FUNCTION_BLOCK LogSchedule (* Basic Function Block Type *)
  (* Standard: 61499-2 *)
  (* Version 0.0, 11/2/2016, chivdan, nxtControl GmbH, Template *)
  PACKAGE Main;
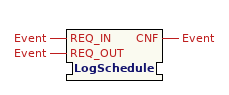
  EVENT_INPUT
    REQ_IN; (* Normal Execution Request *)
    REQ_OUT;
  END_EVENT
  EVENT_OUTPUT
    CNF;
  END_EVENT
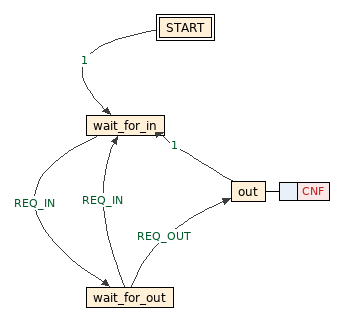
  EC_STATES
    START; (* Initial State *)
    wait_for_in;
    wait_for_out;
    out : -> CNF;
  END_STATES
  EC_TRANSITIONS
    START TO wait_for_in := 1;
    wait_for_in TO wait_for_out := REQ_IN;
    wait_for_out TO out := REQ_OUT;
    out TO wait_for_in := 1;
    wait_for_out TO wait_for_in := REQ_IN;
  END_TRANSITIONS
  ALGORITHM INIT IN ST: (* Initialization algorithm *)
;
  END_ALGORITHM
  ALGORITHM REQ IN ST: (* Normally executed algorithm *)
;
  END_ALGORITHM
END_FUNCTION_BLOCK
